Staubli VAL3: Axis7Status.pgx

public program Axis7Status(bool& x_bPowerOn (dimensions=1), bool& x_bAlarm (dimensions=1), bool& x_bhome (dimensions=1))
begin

  //  x_bAlarm=true
  //  x_bPowerOn=false

  x_bhome=dDio["In4_b7BackHome"]==true
  x_bPowerOn=dDio["In4_b7MotorPower"]==true
  x_bAlarm=dDio["In4_b7MotorError"]==true











end
